FUNCTION makeArray1: ARRAY[0..1] of DINT
VAR_INPUT
    elem0: DINT;
    elem1: DINT;
END_VAR
VAR
    rslt: ARRAY[0..1] of DINT;
END_VAR


        rslt[0] := elem0;
rslt[1] := elem1;
makeArray1 := rslt;

END_FUNCTION

(* stored: ProductVersion 3.1.0.18, Version 1.1.0.1 *)
